(* PLC project M3_13, Desconocido M3_13 1 *)
(* stored: creationDateTime 2025-05-15T11:40:54, modificationDateTime 2025-05-15T13:56:43 *)

PROGRAM Main
  VAR
    xMarcha : BOOL;  (* Marcha de la bomba principal *)
    tTiempoTranscurrido : TIME;  (* Tiempo Transcurrido *)
    xParada : BOOL;  (* Parada de la bomba principal *)
    xBomba : BOOL;  (* Bomba principal *)
    xFalla : BOOL;  (* Falla de la Bomba *)
    xAlertaFalla : BOOL;  (* Alerta de Falla de la Bomba *)
    TON0 : TON;
    TON1 : TON;
  END_VAR

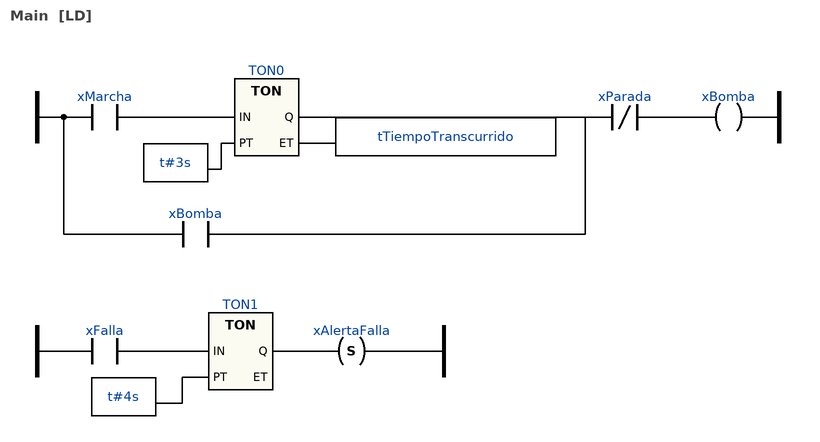
(* LD diagram, written out as Structured Text *)
TON0(IN := xMarcha, PT := t#3s);
xBomba := (xBomba OR TON0.Q) AND NOT xParada;
tTiempoTranscurrido := TON0.ET;
TON1(IN := xFalla, PT := t#4s);
IF TON1.Q THEN xAlertaFalla := TRUE; END_IF;
END_PROGRAM

CONFIGURATION Config0
  RESOURCE Res0 ON PLC
    TASK task0(INTERVAL := T#20ms, PRIORITY := 0);
    PROGRAM instance0 WITH task0 : Main;
  END_RESOURCE
END_CONFIGURATION
